TEXTLIST subinklevel
  1 = 'W1'
  2 = 'W2'
  3 = 'LM1'
  4 = 'LC1'
  5 = 'Y1'
  6 = 'M1'
  7 = 'C1'
  8 = 'K1'
  9 = 'K2'
  10 = 'C2'
  11 = 'M2'
  12 = 'Y2'
  13 = 'LC2'
  14 = 'LM2'
  15 = 'W3'
  16 = 'W4'
   = ''
END_TEXTLIST

(* stored: Version 1.1.0.1, ProductVersion 3.1.4024.11
   TextList subinklevel: Id {8152adf2-8123-406f-94a3-49bdac54e70b} *)
